Fanuc KAREL source: kd00019.KL

PROGRAM KD00019
%STACKSIZE=65535
%PRIORITY=65535
%NOLOCKGROUP
VAR
I : INTEGER
J : INTEGER
B : BOOLEAN
R : REAL
S : STRING[80]
-- UNRESOLVED DECLARATIONS (source type spelling not recovered)
-- REC : TYPE_0x1100 (type_u16=0x1100)
BEGIN
REC.VALUE=1
REC.VALUE=(REC.VALUE + 1)
END KD00019
